(* IEC 61131-3 sources: eCockpitGit/test_project/src/%GVL%GVL_test/%F%GVLFolder/%PRO%PropAlop, 1 file *)

(* ---- %GETSET%Get.st ---- *)
VAR
	temp:BOOL;
END_VAR

(*%!%__DELIMITER__%!%*)
PropAlop		:=		temp AND variablssss;
